// TIA Portal project "s09_security" (V21)

(* hardware
DEVICE "S7-1200 station_1"  S7-1200 Station
   slot 0: "Rack_0"  S7-1200 Rack  Rack  V1.0
   slot 1: "ZZALPHA"  CPU 1212C AC/DC/Rly  6ES7 212-1BD30-0XB0  V2.2
   slot 2: "DI 8x24VDC_1"  SM 1221 DI8 x 24VDC  6ES7 221-1BF30-0XB0  V1.0
DEVICE "S7-1500/ET200MP station_1"  S7-1500 station
   slot 0: "Rail_0"  Rack  6ES7 590-1***0-0AA0
   slot 1: "ZZBRAVO"  CPU 1511-1 PN  6ES7 511-1AK00-0AB0  V1.8
      slot 3: "CPU display_1"  6ES7591-1AA00-0AA0
      slot 32768: "PROFINET interface_1"  X1
         slot 32769: "Port_1"  X1 P1
         slot 32770: "Port_2"  X1 P2
DEVICE "S7-1500/ET200MP station_2"  S7-1500 station
   slot 0: "Rail_0"  Rack  6ES7 590-1***0-0AA0
   slot 1: "ZZCHARLIE"  CPU 1511-1 PN  6ES7 511-1AL03-0AB0  V4.1
      slot 3: "CPU display_1"  6ES7591-1AA00-0AA0
      slot 32768: "PROFINET interface_1"  X1
         slot 32769: "Port_1"  X1 P1
         slot 32770: "Port_2"  X1 P2
      slot 34817: "Virtual CP interface port_1"  Virtual CP interface port  Virtual CP interface port FW V4.1
*)

// ===== PLC "ZZALPHA"  CPU 1212C AC/DC/Rly =====

ORGANIZATION_BLOCK "Main"   // OB1, LAD, ProgramCycle
TITLE = "Main Program Sweep (Cycle)"
{ S7_Optimized_Access := 'TRUE' }
VERSION : 0.1
BEGIN
END_ORGANIZATION_BLOCK

// ===== PLC "ZZBRAVO"  CPU 1511-1 PN =====

VAR_GLOBAL   // PLC tag table "Default tag table"
   "Tag_1" AT %I0.1 : Bool;
   "Tag_2" AT %Q0.2 : Bool;
   "Tag_3" AT %M13.1 : Bool;
   "Tag_4" AT %M12.1 : Bool;
END_VAR

VAR_GLOBAL   // PLC tag table "Tag MyTagTable"
   "Mybool" AT %I0.0 : Bool;   // This is a bolean
   "Mysecondbool" AT %Q0.1 : Bool;
   "MyByte" AT %MB10 : Byte;
   "MyInt" AT %MW20 : Word;
   "MyReal" AT %MD22 : Real;
   "MyDWord" AT %MD26 : DWord;
   "MyTime" AT %MD30 : Time;
   "MyChar" AT %MB34 : Char;   // This is a char
END_VAR

TYPE "User_data_type_1"
   STRUCT
      memberDate : Date := D#1990-01-31;
      memberString : String := 'Hello world';
      memberInt : Int := 7;
      memberBolean : Bool;
   END_STRUCT;
END_TYPE

DATA_BLOCK "DB_Standard"   // DB1
{ S7_Optimized_Access := 'FALSE' }
VERSION : 0.1
   VAR
      my_data_type : "User_data_type_1";
      my_bool : Bool := true;
      my_byte : Byte := 16#4;
      my_int : Int := 5;
      my_dint : DInt := 6;
      my_real : Real := 3.141593;
      my_stringof10 : Array[0..10] of String;
      my_array_of_int : Array[0..3] of Int;
   END_VAR
BEGIN
END_DATA_BLOCK

DATA_BLOCK "DB_Optimized"   // DB2
{ S7_Optimized_Access := 'TRUE' }
VERSION : 0.1
   VAR
      my_data_type : "User_data_type_1";
      my_bool : Bool := true;
      my_byte : Byte := 16#4;
      my_int : Int := 5;
      my_dint : DInt := 6;
      my_real : Real := 3.141593;
      my_sitringof10 : Array[0..10] of String;
      my_array_of_int : Array[0..3] of Int;
   END_VAR
BEGIN
END_DATA_BLOCK

DATA_BLOCK "Block_1_DB"   // DB3
{ S7_Optimized_Access := 'TRUE' }
VERSION : 0.1
// stored: InstanceOfName Block_1
"Block_1"
BEGIN
END_DATA_BLOCK

DATA_BLOCK "Block_2_DB"   // DB4
{ S7_Optimized_Access := 'TRUE' }
VERSION : 0.1
// stored: InstanceOfName Block_2
"Block_2"
BEGIN
END_DATA_BLOCK

FUNCTION_BLOCK "Block_1"   // FB1, FBD
{ S7_Optimized_Access := 'TRUE' }
VERSION : 0.1
   VAR_INPUT
      "M12.1" : Bool;   // My Boolian input
   END_VAR
   VAR_OUTPUT
      "M13.1" : Bool;   // My Boolian output
   END_VAR
   VAR_IN_OUT
      my_inout : Byte := 16#7;   // My IO Byte
   END_VAR
   VAR
      "555" : DInt := 555;
   END_VAR
BEGIN
END_FUNCTION_BLOCK

FUNCTION_BLOCK "Block_2"   // FB2, STL
{ S7_Optimized_Access := 'TRUE' }
VERSION : 0.1
   VAR_INPUT
      MB12 : Byte := 16#3;   // My input byte
   END_VAR
   VAR_OUTPUT
      MB14 : Byte := 16#4;   // My output byte
   END_VAR
   VAR_IN_OUT
      MB15 : Byte;   // My In/Out byte
   END_VAR
   VAR
      "666" : DInt := 666;   // My Static
   END_VAR
BEGIN
END_FUNCTION_BLOCK

ORGANIZATION_BLOCK "Main"   // OB1, LAD, ProgramCycle
TITLE = "Main Program Sweep (Cycle)"
{ S7_Optimized_Access := 'TRUE' }
VERSION : 0.1
   VAR_INPUT
      Initial_Call : Bool;   // Initial call of this OB
      Remanence : Bool;   // =True, if remanent data are available
   END_VAR
BEGIN

REGION Network 1
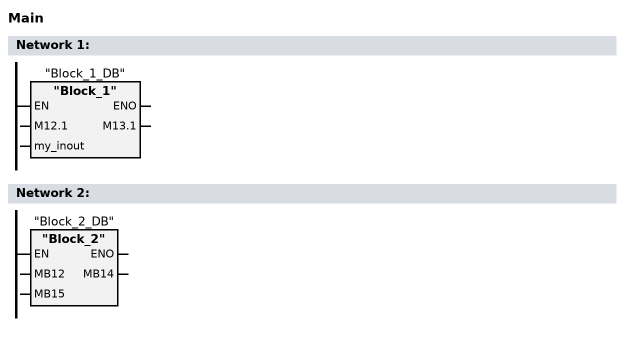
   RUNG wire#powerrail
      "Block_1_DB"("M12.1" :=, my_inout :=, "M13.1" =>)
   END_RUNG
   // the same network as SCL:
   "Block_1_DB"();   // "Block_1"
END_REGION

REGION Network 2
   RUNG wire#powerrail
      "Block_2_DB"(MB12 :=, MB15 :=, MB14 =>)
   END_RUNG
   // the same network as SCL:
   "Block_2_DB"();   // "Block_2"
END_REGION
END_ORGANIZATION_BLOCK

// ===== PLC "ZZCHARLIE"  CPU 1511-1 PN =====

ORGANIZATION_BLOCK "Main"   // OB1, LAD, ProgramCycle
TITLE = "Main Program Sweep (Cycle)"
{ S7_Optimized_Access := 'TRUE' }
VERSION : 0.1
   VAR_INPUT
      Initial_Call : Bool;   // Initial call of this OB
      Remanence : Bool;   // =True, if remanent data are available
   END_VAR
BEGIN
END_ORGANIZATION_BLOCK